FUNCTION_BLOCK burner
  (* Standard: 61499-2 *)
  (* Version 0.1, 2017-00-25, hpea485, UOA *)
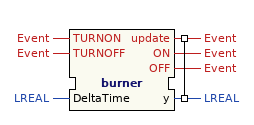
  EVENT_INPUT
    TURNON;
    TURNOFF;
  END_EVENT
  EVENT_OUTPUT
    update WITH y;
    ON;
    OFF;
  END_EVENT
  VAR_INPUT
    DeltaTime : LREAL := 0.01;
  END_VAR
  VAR_OUTPUT
    y : LREAL;
  END_VAR
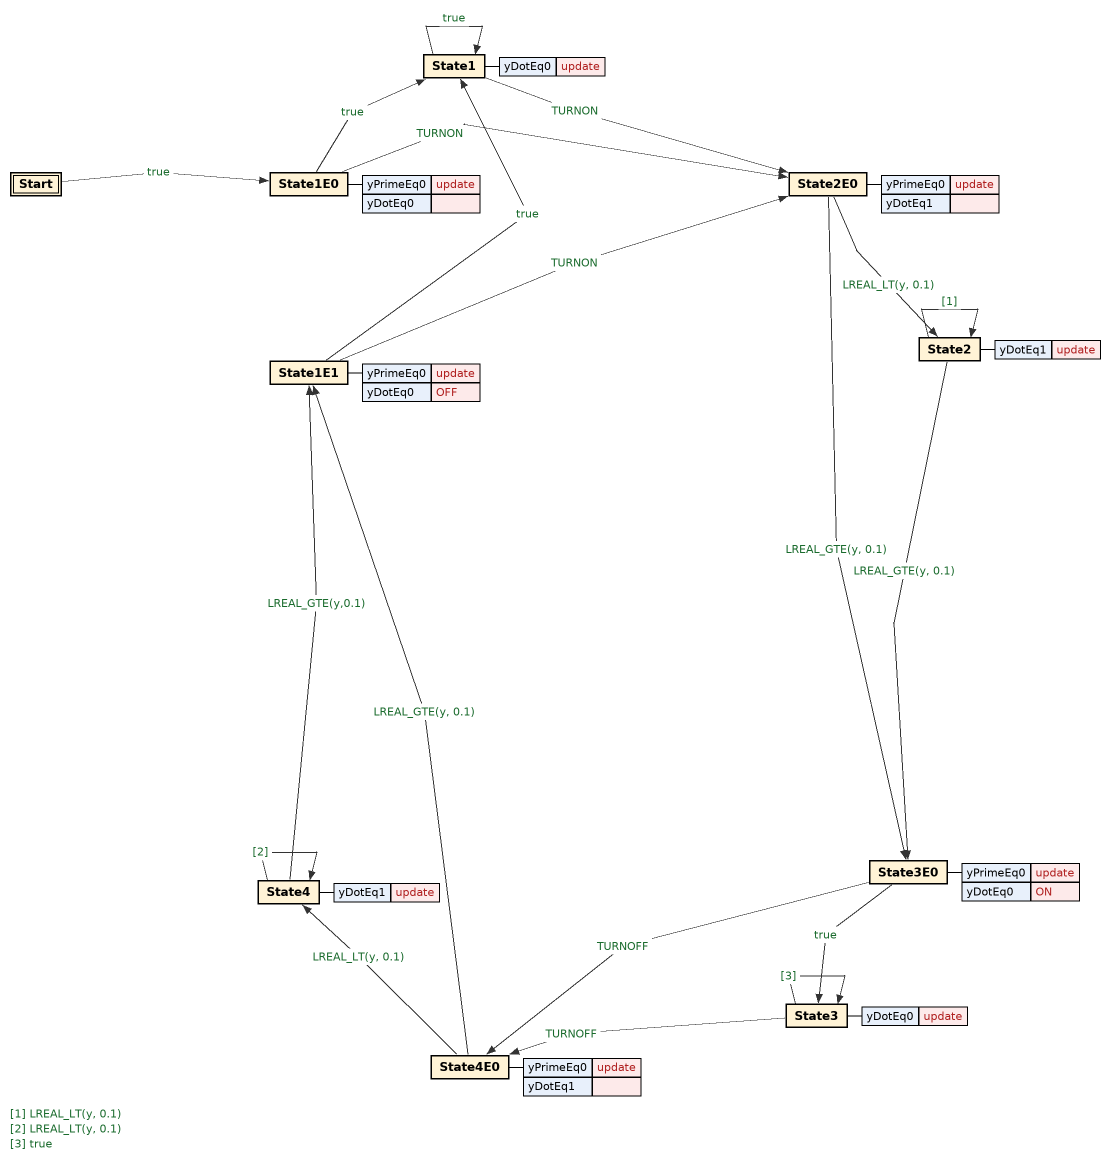
  EC_STATES
    Start;
    State1E0 : yPrimeEq0 -> update, yDotEq0;
    State1 : yDotEq0 -> update;
    State2E0 : yPrimeEq0 -> update, yDotEq1;
    State2 : yDotEq1 -> update;
    State3E0 : yPrimeEq0 -> update, yDotEq0 -> ON;
    State3 : yDotEq0 -> update;
    State4E0 : yPrimeEq0 -> update, yDotEq1;
    State4 : yDotEq1 -> update;
    State1E1 : yPrimeEq0 -> update, yDotEq0 -> OFF;
  END_STATES
  EC_TRANSITIONS
    Start TO State1E0 := true;
    State1E0 TO State2E0 := TURNON;
    State1E0 TO State1 := true;
    State1 TO State2E0 := TURNON;
    State1 TO State1 := true;
    State2E0 TO State3E0 := LREAL_GTE(y, 0.1);
    State2E0 TO State2 := LREAL_LT(y, 0.1);
    State2 TO State3E0 := LREAL_GTE(y, 0.1);
    State2 TO State2 := LREAL_LT(y, 0.1);
    State3E0 TO State4E0 := TURNOFF;
    State3E0 TO State3 := true;
    State3 TO State4E0 := TURNOFF;
    State3 TO State3 := true;
    State4E0 TO State1E1 := LREAL_GTE(y, 0.1);
    State4E0 TO State4 := LREAL_LT(y, 0.1);
    State4 TO State1E1 := LREAL_GTE(y,0.1);
    State4 TO State4 := LREAL_LT(y, 0.1);
    State1E1 TO State2E0 := TURNON;
    State1E1 TO State1 := true;
  END_TRANSITIONS
  ALGORITHM yPrimeEq0 IN C: (* ODE_init *)
y_prime = 0;
  END_ALGORITHM
  ALGORITHM yDotEq0 IN C: (* ODE *)
y_dot = 0;
  END_ALGORITHM
  ALGORITHM yDotEq1 IN C: (* ODE *)
y_dot = 1;
y_trigger = 0.1;
  END_ALGORITHM
END_FUNCTION_BLOCK
